PROGRAM P0_Start_Initialization
VAR
END_VAR

END_PROGRAM

(* stored: Version 1.1.0.1, ProductVersion 3.1.4022.7
   POU P0_Start_Initialization: Id {38462480-6cd7-4fbd-b101-ccb69495903e}, SpecialFunc None *)
